TYPE "udt_FComm"
VERSION : 0.1
// Block: udt_FComm
   STRUCT
      EstopLocal : Bool;
      EstopGlobal : Bool;
      Door_Ok : Bool;
      Door_NormalStop : Bool;
      Door_SafeStop : Bool;
      _05 : Bool;
      LightCurtain_Ok : Bool;
      _07 : Bool;
      _08 : Bool;
      EntryEnable : Bool;
      _10 : Bool;
      _11 : Bool;
      _12 : Bool;
      _13 : Bool;
      _14 : Bool;
      CommOk : Bool;
   END_STRUCT;

END_TYPE
